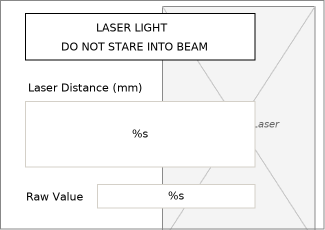
VISUALIZATION V_AI  // 325x230
    Image (162,6 153x236), image: ImagePool.Laser
    Rectangle (25,13 230x47)
    Label (93,20 183x21), "LASER LIGHT"
    Label (58,39 183x21), "DO NOT STARE INTO BEAM"
    Label (25,73 167x30), "Laser Distance (mm)"
    Textfield (25,101 230x66), "%s", text variable: Module_IO.nLaserValue
    Label (23,182 71x30), "Raw Value"
    Textfield (97,184 158x24), "%s", text variable: Laser.nLaserRawValue
END_VISUALIZATION

(* stored: Version 1.1.0.1, ProductVersion 3.1.4024.11
   Visu V_AI: Id {90d1dd3f-7ea7-4b37-9b9d-a863c45849ee} *)
